Yaskawa INFORM job: HOME.JBI

/JOB
//NAME HOME
///FOLDERNAME MASTER
//POS
///NPOS 1,0,0,0,0,0
///TOOL 0
///POSTYPE PULSE
///PULSE
C00000=0,0,0,0,0,0
//INST
///DATE 2021/10/29 11:48
///COMM YMCL HOME POSITION CHECK V1.0
///ATTR SC,RO
///GROUP1 RB1
NOP
'*******************************
'USE THIS JOB TO PLAY OR STEP
'ROBOT TO HOME POSITION TO
'CHECK ALIGNMENT OF HOME
'POSITION ARROWS. DO THIS IF
'MECHANICAL DISPLACEMENT OR LOSS
'OF ABSOLUTE DATA IS SUSPECTED.
'*******************************
MOVJ C00000 VJ=3.12
END
